TYPE RemoteOrder :
STRUCT
	SupplySP: LREAL;
	ExtractSP: LREAL;
	Counter: INT;
	TimeChannels: TimeChannelParameters;
	TemperatureControl: ControllerParameters;
	TemperatureSetPointAdjustment: SetPointAdjustment; 
	SupplyAirControl: ControllerParameters; 
	SupplyAirSetPointAdjustment: SetPointAdjustment; 
	ExtractAirControl: ControllerParameters; 
	ExtractAirSetPointAdjustment: SetPointAdjustment; 
END_STRUCT
END_TYPE

(* stored: Version 1.1.0.1, ProductVersion 3.1.4024.6
   DUT RemoteOrder: Id {7f95e125-9837-42c9-b5b2-3701635a9c02} *)
